PROGRAM MAIN
VAR
END_VAR

//call comunication program

Prg_Server();

END_PROGRAM

(* stored: Version 1.1.0.1, ProductVersion 3.1.4024.9
   POU MAIN: Id {83ade9c1-8e48-4716-845f-723563b17afe}, SpecialFunc None *)
